{attribute 'GeneratedUsingTerminal: EL5001--0000'}
{attribute addProperty BoxType "EL5001--0000"}
{attribute addProperty Id "StatusAT %I*BYTE1ValueAT %I*UDINT4"}
{attribute addProperty CRC "1315168589"}
{attribute addProperty Size "5"}
TYPE Channel_4E63E14D EXTENDS InputBase_8311D824 :
STRUCT
	{attribute addProperty Name "Status"}
	Status AT %I* : BYTE;
	{attribute addProperty Name "Value"}
	Value AT %I* : UDINT;
END_STRUCT
END_TYPE

(* stored: Version 1.2.0.0, ProductVersion 3.1.4024.11
   DUT Channel_4E63E14D: Id {78a5493e-300c-47ff-910a-37e5dda65a7d} *)
